PROGRAM MAIN
VAR
	ErrorString_WithConcat:STRING;
	ErrorString_WithFluentCode:STRING;
	ErrorMessage:STRING := 'Important message';
	ErrorNumber:int := 1;
	_StringBuilder:StringBuilder;
	StringAreEqual:BOOL;
	StringAreStillEqual:BOOL;
END_VAR

ErrorString_WithConcat := CONCAT(CONCAT(CONCAT(CONCAT('Error number: ' , INT_TO_STRING(ErrorNumber)),'. Message: '),ErrorMessage),'.');
ErrorString_WithConcat := Concat('Error number: ' , INT_TO_STRING(ErrorNumber));
ErrorString_WithConcat := Concat(ErrorString_WithConcat , '. Message: ');
ErrorString_WithConcat := Concat(ErrorString_WithConcat , ErrorMessage);
ErrorString_WithConcat := Concat(ErrorString_WithConcat , '.');
							
ErrorString_WithFluentCode := _StringBuilder.Reset()
							.Append('Error number: ')
							.Append(INT_TO_STRING(ErrorNumber))
							.Append('. Message: ')
							.Append(ErrorMessage)
							.Append('.')
							.ToString();
							
StringAreEqual := ErrorString_WithConcat = ErrorString_WithFluentCode;

ErrorString_WithConcat := INSERT( ErrorString_WithConcat, ' extended',43);
ErrorString_WithFluentCode := _StringBuilder.InsertAtLocation(' extended',43).ToString();

StringAreStillEqual :=  ErrorString_WithConcat = ErrorString_WithFluentCode;

END_PROGRAM

(* stored: Version 1.1.0.1, ProductVersion 3.1.4024.0
   POU MAIN: Id {9eec8c03-abcb-4771-a1da-c6b5667fb74a}, SpecialFunc None *)
